FUNCTION_BLOCK FB_SimActuator IMPLEMENTS IActuator
VAR_INPUT
END_VAR
VAR_OUTPUT
END_VAR
VAR
	tmrExtend		: TON;
	tmrRetract		: TON;
	tmrCycle		: TON;
	iExtendDur		: DINT;
	iRetractDur		: DINT;
	
	rand			: DRAND;
	
	bExtended		: BOOL;
	bRetracted		: BOOL;
	
	iCycleState		: DINT;
	STROKE_DUR_MS	: DINT := 2000;
END_VAR

rand(Seed:=TO_INT(iExtendDur + iRetractDur));

METHOD Cycle : BOOL
CASE iCycleState OF
	0:
		IF THIS^.Extend() THEN
			iCycleState := 1;
		END_IF
	1:
		tmrCycle(IN:=TRUE, PT:=T#500MS);
		IF tmrCycle.Q THEN
			tmrCycle(IN:=FALSE);
			iCycleState := 2;
		END_IF
		
	2:
		IF THIS^.Retract() THEN
			iCycleState := 3;
		END_IF
		
	3:
		iCycleState := 0;
		Cycle := TRUE;
END_CASE
END_METHOD

METHOD Extend : BOOL
IF NOT tmrExtend.IN THEN
	bRetracted := FALSE;
	iExtendDur := TO_DINT(rand.Num * 1000) + STROKE_DUR_MS;
	tmrExtend(PT:=DINT_TO_TIME(iExtendDur)); 	
END_IF

IF tmrExtend.Q THEN
	tmrExtend(IN:=FALSE);
	bExtended := TRUE;
	Extend := TRUE;
ELSE
	tmrExtend(IN:=TRUE);
	Extend := FALSE;
END_IF
END_METHOD

PROPERTY Extended : BOOL
GET
Extended := bExtended;
END_GET
END_PROPERTY

METHOD Retract : BOOL
IF NOT tmrRetract.IN THEN
	bExtended := FALSE;
	iRetractDur := TO_DINT(rand.Num * 1000) + STROKE_DUR_MS;
	tmrRetract(PT:=DINT_TO_TIME(iRetractDur)); 	
END_IF

IF tmrRetract.Q THEN
	bRetracted := TRUE;
	tmrRetract(IN:=FALSE);
	Retract := TRUE;
ELSE
	tmrRetract(IN:=TRUE);
	Retract := FALSE;
END_IF
END_METHOD

PROPERTY Retracted : BOOL
GET
Retracted := bRetracted;
END_GET
END_PROPERTY

END_FUNCTION_BLOCK

(* stored: Version 1.1.0.1, ProductVersion 3.1.4024.12
   POU FB_SimActuator: Id {b60feaab-d854-40dc-b58d-c92ca4bd5a91}, SpecialFunc None
   Method Cycle: Id {37965100-d96c-4645-8c71-ca1df0408b13}
   Method Extend: Id {40a95e29-a632-41af-a987-4c935a3fa911}
   Property Extended: Id {b8ac5087-3ff2-43a7-b584-1f32518f4381}
   Get Get: Id {adb61051-46e0-4181-8afd-273eaf7161cb}
   Method Retract: Id {55bc305c-9eba-4946-bab0-3b5fb897cca8}
   Property Retracted: Id {9945b710-2862-4e2a-92dd-863f037f83ee}
   Get Get: Id {52d1f740-9588-4293-91ea-6e94a1c38ca8} *)
